// TIA Portal V16 export
// export: Created 2024-09-05T17:40:15.0634235Z, ExportSetting WithDefaults, DisplayName Totally Integrated Automation Portal, DisplayVersion V16 Update 6, DisplayName TIA Portal Version Control Interface, DisplayVersion V16 Update 2, DisplayName TIA Portal Openness, DisplayVersion V16 Update 6, DisplayName STEP 7 Professional, DisplayVersion V16 Update 6, DisplayName STEP 7 Safety, DisplayVersion V16, DisplayName WinCC Advanced, DisplayVersion V16 Update 6
TYPE "UDT_FittingStatus"
// stored: IsFailsafeCompliant false
   STRUCT
      Start : Bool;
      Done : Bool;
      Running : Bool;
      Returning : Bool;
      OK : Bool;
      ContinueFitting : Bool;
      ContinueReturn : Bool;
      InPreposition : Bool;
      continueWithSupportToWork : Bool;
      StartSequence : Bool;
      DoneSequence : Bool;
      PartErrors : Array[1..8] of Bool;
      rivetStatus : SInt;
   END_STRUCT;
END_TYPE
